(* IEC 61131-3 sources: programs/VI-54/VI-54_20171205/VI-54_20171205/Stations/Screen/LseClass170718/Class/LasalBuiltDate, 1 file *)

(* ---- LasalBuiltDate.st ---- *)
(*!
<Class
	Name               = "LasalBuiltDate"
	Revision           = "0.0"
	RealtimeTask       = "false"
	CyclicTask         = "false"
	BackgroundTask     = "false"
	Sigmatek           = "false"
	OSInterface        = "false"
	HighPriority       = "false"
	Automatic          = "false"
	UpdateMode         = "Prescan"
	SharedCommandTable = "true"
	Objectsize         = "(660,180)">
	<Channels>
		<Server Name="Datum" Visualized="false" Initialize="false" WriteProtected="false" Retentive="false"/>
		<Client Name="filesys" Required="false" Internal="false"/>
		<Client Name="ToLasalBuiltString" Required="true" Internal="false"/>
	</Channels>
	<Network Name="LasalBuiltDate">
		<!-- List of Components in this network -->
		<Components>
			<Object
				Name       = "_base"
				Class      = "String"
				Position   = "(218,120)"
				Visualized = "false">
				<Channels>
					<Server Name="Data"/>
					<Client Name="SingleRealloc" Value="1"/>
				</Channels>
			</Object>
		</Components>
		<Comments>
		</Comments>
		<!-- List of Connections in this network -->
		<Connections>
			<Connection Source="this.Data" Destination="_base.Data" Vertices="(946,210),(774,210),"/>
		</Connections>
		<!-- Headerfiles -->
		<Options>
		</Options>
	</Network>
</Class>
*)
#pragma using String

LasalBuiltDate : CLASS
: String
  //Servers:
	Datum 	: SvrCh__DDE_DATIM;
  //Clients:
	filesys 	: CltChCmd__FileSys;
	ToLasalBuiltString 	: CltChCmd_String;
  //Variables:
		Fileinfo 	: _DDE_INFO;
		Vnr : ARRAY [0..10] OF CHAR;

		DateStruct 	: DateTime;
		udDatum 	: _DDE_DATIM;
  //Functions:

	FUNCTION VIRTUAL GLOBAL Init;

	FUNCTION ConvToDate
		VAR_INPUT
			dde_dt 	: _DDE_DATIM;
		END_VAR
		VAR_OUTPUT
			DT_struct 	: DateTime;
		END_VAR;

	FUNCTION VIRTUAL GLOBAL Datum::Read
		VAR_OUTPUT
			output (EAX) 	: _DDE_DATIM;
		END_VAR;

	FUNCTION VIRTUAL GLOBAL Datum::Write
		VAR_INPUT
			input (EAX) 	: _DDE_DATIM;
		END_VAR
		VAR_OUTPUT
			result (EAX) 	: _DDE_DATIM;
		END_VAR;
  //Tables:
	FUNCTION @STD
		VAR_OUTPUT
			ret_code	: CONFSTATES;
		END_VAR;
	FUNCTION GLOBAL TAB @CT_;
END_CLASS;

#pragma usingLtd _FileSys

FUNCTION VIRTUAL GLOBAL LasalBuiltDate::Init

  FileSys.FindFirst("c:\lslwork\","project.lob",#FileInfo,0,0);

  udDatum:=Fileinfo.datetime;

  DateStruct:=ConvToDate(udDatum);

  Datum:=udDatum;

  ToLasalBuiltString.writedataoff(20,0,#DateStruct.str[0]);

END_FUNCTION

FUNCTION VIRTUAL GLOBAL LasalBuiltDate::Datum::Read
	VAR_OUTPUT
		output (EAX) 	: _DDE_DATIM;
	END_VAR

	output := Datum;

END_FUNCTION

FUNCTION VIRTUAL GLOBAL LasalBuiltDate::Datum::Write
	VAR_INPUT
		input (EAX) 	: _DDE_DATIM;
	END_VAR
	VAR_OUTPUT
		result (EAX) 	: _DDE_DATIM;
	END_VAR

	Datum := input;
 	result := Datum;

END_FUNCTION

FUNCTION LasalBuiltDate::ConvToDate
	VAR_INPUT
		dde_dt 	: _DDE_DATIM;
	END_VAR
	VAR_OUTPUT
		DT_struct 	: DateTime;
	END_VAR
  VAR
    dde_udint:udint;
  END_VAR;

  dde_udint:=dde_dt$udint;

  // read date time data

  DT_struct.Year    := (dde_udint AND 2#11111110000000000000000000000000) shr 25;

  DT_struct.Year    += 1980;

  DT_struct.Month   := (dde_udint AND 2#00000001111000000000000000000000) shr 21;

  DT_struct.Day     :=   (dde_udint AND 2#00000000000111110000000000000000) shr 16;

  DT_struct.Hour    := (dde_udint AND 2#00000000000000001111100000000000) shr 11;

  DT_struct.Minute  := (dde_udint AND 2#00000000000000000000011111100000) shr 5;

  //write date time data in a string

  if DT_struct.Day < 10 then

     DtoA(#dt_struct.str[1],to_DINT(DT_struct.Day), 0x0800,sizeof(_ASCII));

     dt_struct.str[0] := '0';

  else

     DtoA(#dt_struct.str[0],to_DINT(DT_struct.Day), 0x0800,sizeof(_ASCII));

  end_if;

  dt_struct.str[2] := '.';

  if DT_struct.Month < 10 then

     DtoA(#dt_struct.str[4],to_DINT(DT_struct.Month), 0x0800,sizeof(_ASCII));

     dt_struct.str[3] := '0';

  else

     DtoA(#dt_struct.str[3],to_DINT(DT_struct.Month), 0x0800,sizeof(_ASCII));

  end_if;

  dt_struct.str[5] := '.';

  DtoA(#dt_struct.str[6],to_DINT(DT_struct.Year), 0x0800,sizeof(_ASCII));

  dt_struct.str[10] := 32;

  dt_struct.str[11] := 32;

  if DT_struct.Hour < 10 then

     DtoA(#dt_struct.str[13],to_DINT(DT_struct.Hour), 0x0800,sizeof(_ASCII));

     dt_struct.str[12] := '0';

  else

     DtoA(#dt_struct.str[12],to_DINT(DT_struct.Hour), 0x0800,sizeof(_ASCII));

  end_if;

  dt_struct.str[14] := ':';

  if DT_struct.Minute < 10 then

     DtoA(#dt_struct.str[16],to_DINT(DT_struct.Minute), 0x0800,sizeof(_ASCII));

     dt_struct.str[15] := '0';

  else

     DtoA(#dt_struct.str[15],to_DINT(DT_struct.Minute), 0x0800,sizeof(_ASCII));

  end_if;

  dt_struct.str[17] := 0;

END_FUNCTION
